Omron CX-Programmer project NewProject (CX-Programmer 9.70)

# PLC NewPLC1: CJ1M CPU11

## Program NewProgram1 (cyclic task 0)
Local symbols
A BOOL
B BOOL
O BOOL

### Section NxN

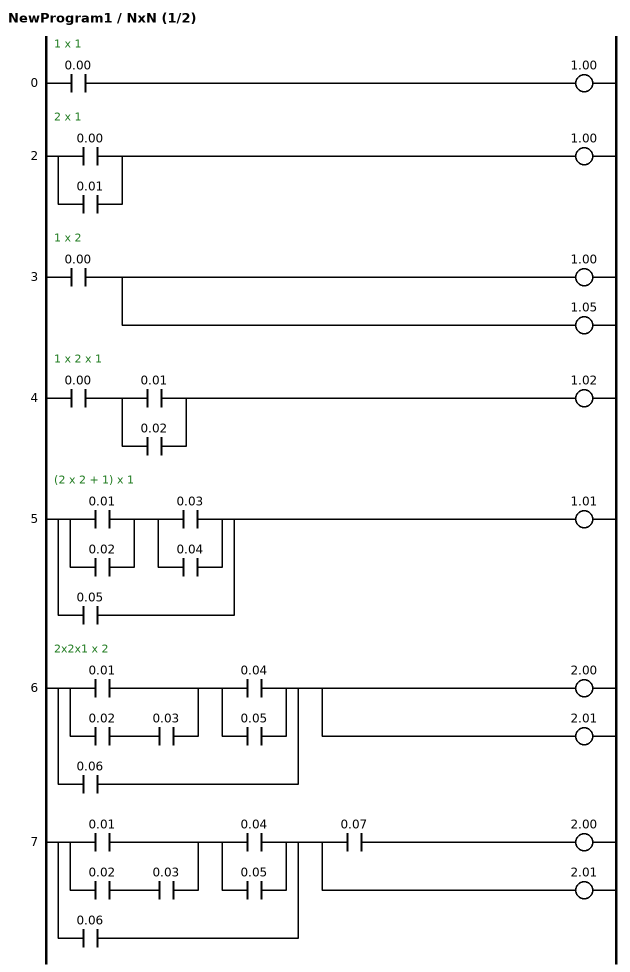
; rung 0: 1 x 1
LD 0.00
OUT 1.00
; rung 2: 2 x 1
LD 0.00
OR 0.01
OUT 1.00
; rung 3: 1 x 2
LD 0.00
OUT 1.00
OUT 1.05
; rung 4: 1 x 2 x 1
LD 0.00
LD 0.01
OR 0.02
ANDLD
OUT 1.02
; rung 5: (2 x 2 + 1) x 1
LD 0.01
OR 0.02
LD 0.03
OR 0.04
ANDLD
OR 0.05
OUT 1.01
; rung 6: 2x2x1 x 2
LD 0.01
LD 0.02
AND 0.03
ORLD
LD 0.04
OR 0.05
ANDLD
OR 0.06
OUT 2.00
OUT 2.01
; rung 7
LD 0.01
LD 0.02
AND 0.03
ORLD
LD 0.04
OR 0.05
ANDLD
OR 0.06
OUT TR0
AND 0.07
OUT 2.00
LD TR0
OUT 2.01

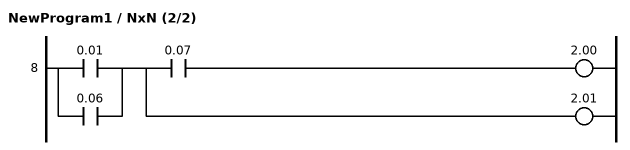
; rung 8
LD 0.01
OR 0.06
OUT TR0
AND 0.07
OUT 2.00
LD TR0
OUT 2.01

### Section 연습

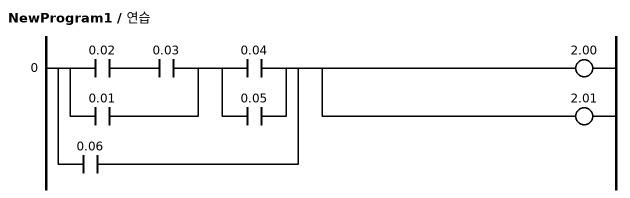
; rung 0
LD 0.02
AND 0.03
LD 0.01
ORLD
LD 0.04
LD 0.05
ORLD
ANDLD
LD 0.06
ORLD
OUT 2.00
OUT 2.01

### Section END
; rung 0
END(001)